{attribute 'GeneratedUsingTerminal: EL5002-0000-0016'}
{attribute addProperty BoxType "EL5002-0000-0016"}
{attribute addProperty Id "EtcSlaveTerminalBaseSSI_Inputs_Channel_1AT %I*SSI_Inputs_Channel_0E3D8E3310SSI_Inputs_Channel_2AT %I*SSI_Inputs_Channel_0E3D8E3310WcStateAT %I*WcState_9091E0EB2InfoDataAT %I*InfoData_32EB74EA10"}
{attribute addProperty CRC "2169208955"}
{attribute addProperty Size "32"}
TYPE EL5002_814B807B EXTENDS EtcSlaveTerminalBase :
STRUCT
	{attribute addProperty Name "SSI_Inputs_Channel_1"}
	SSI_Inputs_Channel_1 : SSI_Inputs_Channel_0E3D8E33;
	{attribute addProperty Name "SSI_Inputs_Channel_2"}
	SSI_Inputs_Channel_2 : SSI_Inputs_Channel_0E3D8E33;
	{attribute addProperty Name "WcState"}
	WcState : WcState_9091E0EB;
	{attribute addProperty Name "InfoData"}
	InfoData : InfoData_32EB74EA;
END_STRUCT
END_TYPE

(* stored: Version 1.2.0.0, ProductVersion 3.1.4024.9
   DUT EL5002_814B807B: Id {e303eeed-d622-4911-9868-29580a3f5c71} *)
